(* PLC project CoDeSys External Library Template, WAGO e!COCKPIT e!COCKPIT, author 3S - Smart Software Solutions GmbH *)
(* stored: creationDateTime 2019-10-29T12:37:19.8905021, version 3.5.5.30, modificationDateTime 2019-10-29T12:36:39.3744516, organization 3S - Smart Software Solutions GmbH *)
(* Library project template with all possible element types, docu and a sample project structure *)

FUNCTION fnKomunikatMACAdres : STRING
  VAR_INPUT
    sKomunikat : alSTRINGKomunikat;
  END_VAR
  VAR
    typKomunikat : typKomunikat;
    intBlad : INT;
  END_VAR

            fnKomunikatInOut(	xStringNaStrukture := TRUE ,
					xStringUpdateZeStruktury := FALSE ,
					xStrukturyNaString := FALSE ,
					xWyczyscStrukture := FALSE ,
					xAktualizujZnacznikCzasu := FALSE ,
					xAktualizujDlugoscDanych := FALSE ,
					sKomunikat := sKomunikat ,
					typKomunikat := typKomunikat ,
					intBlad := intBlad);

fnKomunikatMACAdres := typKomunikat.sMACAdres;

          
END_FUNCTION
